// Mitsubishi GX Works2 project: PLChigh03   PLC: Q02U

PROGRAM MAIN
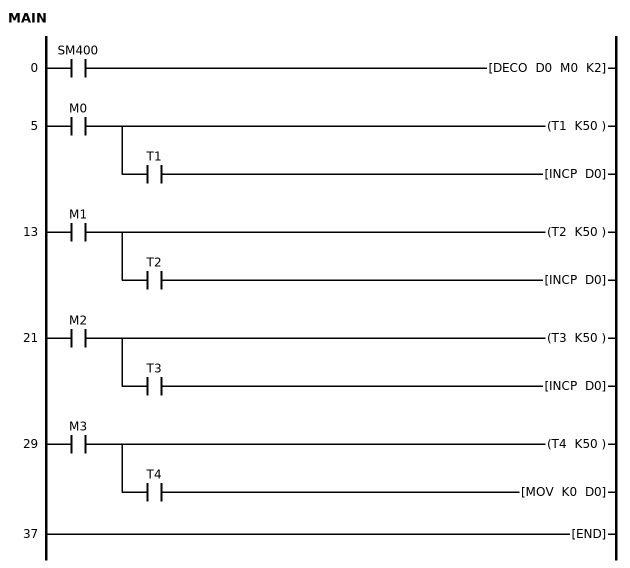
0     LD      SM400
      DECO    D0 M0 K2
5     LD      M0
      OUT     T1 K50
      AND     T1
      INCP    D0
13    LD      M1
      OUT     T2 K50
      AND     T2
      INCP    D0
21    LD      M2
      OUT     T3 K50
      AND     T3
      INCP    D0
29    LD      M3
      OUT     T4 K50
      AND     T4
      MOV     K0 D0
37    END
END_PROGRAM
